TYPE StatsFaultFIFOBuffer :
STRUCT
	Size: UDINT := 500;
	Buffer: ARRAY [0..499] OF StatsFault;
END_STRUCT
END_TYPE

(* stored: Version 1.1.0.1, ProductVersion 3.1.4024.9
   DUT StatsFaultFIFOBuffer: Id {0838f956-3e44-4d27-848d-90e48cadbd48} *)
